// TwinCAT 3 PLC project PLC_1
// ProgramVersion: 3.1.4024.0
// libraries:
//   Tc2_MC2, * (Beckhoff Automation GmbH)
//   Tc2_Standard, * (Beckhoff Automation GmbH)
//   Tc2_System, * (Beckhoff Automation GmbH)
//   Tc3_IotBase, * (Beckhoff Automation GmbH)
//   Tc3_JsonXml, * (Beckhoff Automation GmbH)
//   Tc3_Module, * (Beckhoff Automation GmbH)
// project tree:
//   DUTs/ E_MC.TcDUT
//   GVLs/ GVL_PLC.TcGVL
//   / PlcTask.TcTTO
//   POUs/ FB_Sequence.TcPOU, FB_MQTT.TcPOU, MAIN.TcPOU
// real-time tasks:
//   TASK PlcTask: cycle T#10ms, priority 20, ADS port 350
// motion (NC):
//   TASK NC-Task 1 SAF: cycle T#2ms, priority 4, ADS port 501
//   TASK NC-Task 1 SVB: cycle T#10ms, priority 8, ADS port 511
//   AXIS StepAxis (id 1)
//     General: UnitName=Degree
//     Dynamic: Acceleration=727.2, Deceleration=727.2, Jerk=14689.4
//     Velo: Maximum=3600
//     PositionAreaControl: Enable=false
//     TargetPosControl: Enable=false
//     OtherSettings: AllowMotionCmdToSlave=true
//     encoder EncType=4
//       EncPara: ScaleFactorNumerator=0.028125, MaxCount=#x0000ffff
//         Inc: RefMode=2, RefSoftSyncMask=#x0000ffff
//     drive DrvType=24
//       Analog: VeloReferenz=3600, VeloScale=32, TorqueSetpointScale=10, ScaleFactorActTorque=0.1
//       TimeComp: TaskDelayCycles=1
//     controller CtrType=1
//       CtrPara: PriorControlFactor=1
//         PosDiffControl: Enable=false
//         PID: PosKp=3.5
//         Observer: BandWidth=20
//   AXIS Axis 2 (id 2)
//     OtherSettings: AllowMotionCmdToSlave=true
//     encoder EncType=4
//       EncPara: MaxCount=#x0000ffff
//         Inc: RefSoftSyncMask=#x0000ffff
//     drive DrvType=24
//       Analog: TorqueSetpointScale=10, ScaleFactorActTorque=0.1
//       TimeComp: TaskDelayCycles=1
//     controller CtrType=1
//       CtrPara: PriorControlFactor=1
//         Observer: BandWidth=20
//   AXIS ServoAxis (id 3)
//     General: UnitName=Degree
//     Dynamic: Acceleration=200, Deceleration=200, Jerk=100
//     Velo: Maximum=12000
//     PositionAreaControl: Enable=false
//     TargetPosControl: Enable=false
//     OtherSettings: AllowMotionCmdToSlave=true
//     encoder EncType=19
//       EncPara: ScaleFactorNumerator=0.000343322753906, MaxCount=#xffffffff
//     drive DrvType=16
//       DrvPara: MaxCount=#xffffffff, DriveControlDWord=#x00020000
//         Analog: VeloReferenz=12000, VeloScale=32, TorqueSetpointScale=10, ScaleFactorActTorque=0.1
//         TimeComp: TaskDelayCycles=1
//     controller CtrType=1
//       CtrPara: PriorControlFactor=1
//         PosDiffControl: Enable=false
//         Observer: BandWidth=20
// I/O:
//   DEVICE Device 3 (EtherCAT), AmsNetId 192.168.99.3.4.1
//     Term 1 (EK1100) [EK1100 EtherCAT Coupler (2A E-Bus)]
//       Term 2 (EL1008) [EL1008 8Ch. Dig. Input 24V, 3ms]
//       Term 3 (EL1008) [EL1008 8Ch. Dig. Input 24V, 3ms]
//       Term 4 (EL2008) [EL2008 8Ch. Dig. Output 24V, 0.5A]
//       Term 5 (EL2624) [EL2624 4Ch. Relay Output, NO (125V AC / 30V DC)]
//       Term 6 (EL6001) [EL6001 Interface (RS232)]
//       Term 15 (EL9011) [EL9011 End Terminal]
//     Term 7 (EK1100) [EK1100 EtherCAT Coupler (2A E-Bus)]
//       Term 8 (EL7031-0030) [EL7031-0030 1Ch. Stepper motor output stage (24V, 2.8A)]
//       Term 9 (EL6070-0033) [EL6070-0033 1Ch. Licence key terminal, individual licences]
//       Term 10 (EL7031-0030) [EL7031-0030 1Ch. Stepper motor output stage (24V, 2.8A)]
//       Term 16 (EL9011) [EL9011 End Terminal]
//     Term 11 (EK1818) [EK1818 EtherCAT IO-Coupler  (1A E-Bus, 8 Ch. Dig. In, 3ms, 4 Ch. Dig. Out 24V, 0,5A)]
//       Term 12 (EL7211-9014) [EL7211-9014 1Ch. MDP742 Servo motor output stage with OCT (50V, 4.5A RMS) and STO input]
//       Term 13 (EL1918) [EL1918, 8Ch. Safety Input 24V, TwinSAFE]
//         modules: Module 1 (FSOE), Module 2 (FSLOGIC)
//       Term 14 (EL3208) [EL3208 8Ch. Ana. Input PT100 (RTD)]
//       Term 17 (EL9011) [EL9011 End Terminal]
//   DEVICE Device 2 (RT-Ethernet Protocol), AmsNetId 192.168.99.3.3.1
// variable links:
//   NC-Task 1 SAF/Axes/Axis 2 <-> Device 3 (EtherCAT)/Term 7 (EK1100)/Term 10 (EL7031-0030)
//     Drive/Inputs/In/nState1 @bit 3 <-> STM Status/Status/Error
//     Drive/Inputs/In/nState1 @bit 5 <-> STM Status/Status/Moving negative
//     Drive/Inputs/In/nState1 @bit 4 <-> STM Status/Status/Moving positive
//     Drive/Inputs/In/nState1 @bit 1 <-> STM Status/Status/Ready
//     Drive/Inputs/In/nState1 <-> STM Status/Status/Ready to enable
//     Drive/Inputs/In/nState1 @bit 6 <-> STM Status/Status/Torque reduced
//     Drive/Inputs/In/nState1 @bit 2 <-> STM Status/Status/Warning
//     Drive/Inputs/In/nState2 @bit 3 <-> STM Status/Status/Digital input 1
//     Drive/Inputs/In/nState2 @bit 4 <-> STM Status/Status/Digital input 2
//     Drive/Inputs/In/nState2 @bit 5 <-> STM Status/Status/Sync error
//     Drive/Inputs/In/nState2 @bit 7 <-> STM Status/Status/TxPDO Toggle
//     Drive/Inputs/In/nState4 @bit 1 <-> WcState/InputToggle
//     Drive/Inputs/In/nState4 <-> WcState/WcState
//     Drive/Outputs/Out/nCtrl1 <-> STM Control/Control/Enable
//     Drive/Outputs/Out/nCtrl1 @bit 2 <-> STM Control/Control/Reduce torque
//     Drive/Outputs/Out/nCtrl1 @bit 1 <-> STM Control/Control/Reset
//     Drive/Outputs/Out/nDataOut2[0] <-> STM Velocity/Velocity
//     Enc/Inputs/In/nDataIn1[0] <-> ENC Status compact/Counter value
//     Enc/Inputs/In/nDataIn2[0] <-> ENC Status compact/Latch value
//     Enc/Inputs/In/nState1 @bit 4 <-> ENC Status compact/Status/Counter overflow
//     Enc/Inputs/In/nState1 @bit 3 <-> ENC Status compact/Status/Counter underflow
//     Enc/Inputs/In/nState1 @bit 1 <-> ENC Status compact/Status/Latch extern valid
//     Enc/Inputs/In/nState1 @bit 2 <-> ENC Status compact/Status/Set counter done
//     Enc/Inputs/In/nState2 @bit 4 <-> ENC Status compact/Status/Status of extern latch
//     Enc/Inputs/In/nState2 @bit 5 <-> ENC Status compact/Status/Sync error
//     Enc/Inputs/In/nState2 @bit 7 <-> ENC Status compact/Status/TxPDO Toggle
//     Enc/Inputs/In/nState4 @bit 1 <-> WcState/InputToggle
//     Enc/Inputs/In/nState4 <-> WcState/WcState
//     Enc/Outputs/Out/nCtrl1 @bit 3 <-> ENC Control compact/Control/Enable latch extern on negative edge
//     Enc/Outputs/Out/nCtrl1 @bit 1 <-> ENC Control compact/Control/Enable latch extern on positive edge
//     Enc/Outputs/Out/nCtrl1 @bit 2 <-> ENC Control compact/Control/Set counter
//     Enc/Outputs/Out/nDataOut1[0] <-> ENC Control compact/Set counter value
//   NC-Task 1 SAF/Axes/ServoAxis <-> Device 3 (EtherCAT)/Term 11 (EK1818)/Term 12 (EL7211-9014)
//     Drive/Inputs/In/nDcOutputTime <-> InfoData/DcOutputShift
//     Drive/Inputs/In/nState1 <-> DRV Statusword/Statusword
//     Drive/Inputs/In/nState2 <-> DRV Statusword/Statusword @bit 8
//     Drive/Inputs/In/nState4 @bit 1 <-> WcState/InputToggle
//     Drive/Inputs/In/nState4 <-> WcState/WcState
//     Drive/Outputs/Out/nCtrl1 <-> DRV Controlword/Controlword
//     Drive/Outputs/Out/nCtrl2 <-> DRV Controlword/Controlword @bit 8
//     Drive/Outputs/Out/nDataOut2 <-> DRV Target velocity/Target velocity
//     Enc/Inputs/In/nDataIn1 <-> FB Position/Position
//     Enc/Inputs/In/nDcInputTime <-> InfoData/DcInputShift
//     Enc/Inputs/In/nState4 @bit 1 <-> WcState/InputToggle
//     Enc/Inputs/In/nState4 <-> WcState/WcState
//   NC-Task 1 SAF/Axes/StepAxis <-> Device 3 (EtherCAT)/Term 7 (EK1100)/Term 8 (EL7031-0030)
//     Drive/Inputs/In/nState1 @bit 3 <-> STM Status/Status/Error
//     Drive/Inputs/In/nState1 @bit 5 <-> STM Status/Status/Moving negative
//     Drive/Inputs/In/nState1 @bit 4 <-> STM Status/Status/Moving positive
//     Drive/Inputs/In/nState1 @bit 1 <-> STM Status/Status/Ready
//     Drive/Inputs/In/nState1 <-> STM Status/Status/Ready to enable
//     Drive/Inputs/In/nState1 @bit 6 <-> STM Status/Status/Torque reduced
//     Drive/Inputs/In/nState1 @bit 2 <-> STM Status/Status/Warning
//     Drive/Inputs/In/nState2 @bit 3 <-> STM Status/Status/Digital input 1
//     Drive/Inputs/In/nState2 @bit 4 <-> STM Status/Status/Digital input 2
//     Drive/Inputs/In/nState2 @bit 5 <-> STM Status/Status/Sync error
//     Drive/Inputs/In/nState2 @bit 7 <-> STM Status/Status/TxPDO Toggle
//     Drive/Inputs/In/nState4 @bit 1 <-> WcState/InputToggle
//     Drive/Inputs/In/nState4 <-> WcState/WcState
//     Drive/Outputs/Out/nCtrl1 <-> STM Control/Control/Enable
//     Drive/Outputs/Out/nCtrl1 @bit 2 <-> STM Control/Control/Reduce torque
//     Drive/Outputs/Out/nCtrl1 @bit 1 <-> STM Control/Control/Reset
//     Drive/Outputs/Out/nDataOut2[0] <-> STM Velocity/Velocity
//     Enc/Inputs/In/nDataIn1[0] <-> ENC Status compact/Counter value
//     Enc/Inputs/In/nDataIn2[0] <-> ENC Status compact/Latch value
//     Enc/Inputs/In/nState1 @bit 4 <-> ENC Status compact/Status/Counter overflow
//     Enc/Inputs/In/nState1 @bit 3 <-> ENC Status compact/Status/Counter underflow
//     Enc/Inputs/In/nState1 @bit 1 <-> ENC Status compact/Status/Latch extern valid
//     Enc/Inputs/In/nState1 @bit 2 <-> ENC Status compact/Status/Set counter done
//     Enc/Inputs/In/nState2 @bit 4 <-> ENC Status compact/Status/Status of extern latch
//     Enc/Inputs/In/nState2 @bit 5 <-> ENC Status compact/Status/Sync error
//     Enc/Inputs/In/nState2 @bit 7 <-> ENC Status compact/Status/TxPDO Toggle
//     Enc/Inputs/In/nState4 @bit 1 <-> WcState/InputToggle
//     Enc/Inputs/In/nState4 <-> WcState/WcState
//     Enc/Outputs/Out/nCtrl1 @bit 3 <-> ENC Control compact/Control/Enable latch extern on negative edge
//     Enc/Outputs/Out/nCtrl1 @bit 1 <-> ENC Control compact/Control/Enable latch extern on positive edge
//     Enc/Outputs/Out/nCtrl1 @bit 2 <-> ENC Control compact/Control/Set counter
//     Enc/Outputs/Out/nDataOut1[0] <-> ENC Control compact/Set counter value
//   PLC_1/PLC_1 Instance <-> Device 2 (RT-Ethernet Protocol)
//     PlcTask Inputs/GVL_PLC.uiDevState <-> Inputs/DevState
//   PLC_1/PLC_1 Instance <-> Device 3 (EtherCAT)/Term 1 (EK1100)/Term 2 (EL1008)
//     PlcTask Inputs/MAIN.fbSequence.xButton_NO3 <-> Channel 1/Input
//   PLC_1/PLC_1 Instance <-> Device 3 (EtherCAT)/Term 1 (EK1100)/Term 3 (EL1008)
//     PlcTask Inputs/MAIN.fbSequence.xButton_NO1 <-> Channel 2/Input
//     PlcTask Inputs/MAIN.fbSequence.xButton_NO2 <-> Channel 7/Input
//   PLC_1/PLC_1 Instance <-> NC-Task 1 SAF/Axes/ServoAxis
//     PlcTask Inputs/MAIN.ServoAxis.NcToPlc <-> Outputs/ToPlc
//     PlcTask Outputs/MAIN.ServoAxis.PlcToNc <-> Inputs/FromPlc
//   PLC_1/PLC_1 Instance <-> NC-Task 1 SAF/Axes/StepAxis
//     PlcTask Inputs/MAIN.StepAxis.NcToPlc <-> Outputs/ToPlc
//     PlcTask Outputs/MAIN.StepAxis.PlcToNc <-> Inputs/FromPlc

CONFIGURATION PLC_1
    RESOURCE PLC ON TwinCAT3
        TASK PlcTask(INTERVAL := T#10ms, PRIORITY := 20);
        PROGRAM MAIN WITH PlcTask : MAIN;
    END_RESOURCE
END_CONFIGURATION

// ---- DUTs/E_MC.TcDUT
{attribute 'qualified_only'}
{attribute 'strict'}
TYPE E_MC :
(
	Idle,
	
	RestartCall,
	RestartEffect,
	PowerCall,
	PowerEffect,
	
	HomingCallStep,   
	HomingEffectStep,
	HomingCallServo,   
	HomingEffectServo,
	Execute,
	
	CoupleCallStepMaster,
	CoupleEffectStepMaster,
	MoveAbsCallStepMaster,
	MoveAbsEffectStepMaster,
	DecoupleCallStepMaster,
	DecoupleEffectStepMaster,
	
	
	CoupleCallServoMaster,
	CoupleEffectServoMaster,
	MoveAbsCallServoMaster,
	MoveAbsEffectServoMaster,
	DecoupleCallServoMaster,
	DecoupleEffectServoMaster,
	
	DecoupleCallOnReset,
	DecoupleEffectOnReset,	
	RestartCallOnReset,
	RestartEffectOnReset,	
	
	Error
);
END_TYPE

// ---- GVLs/GVL_PLC.TcGVL
{attribute 'qualified_only'}
VAR_GLOBAL
	lrActPosition	:	LREAL;
	uiDevState	AT%I*	:	UINT;
END_VAR

// ---- POUs/MAIN.TcPOU
PROGRAM MAIN
VAR
	StepAxis	:	AXIS_REF;
	ServoAxis	:	AXIS_REF;
	fbMqtt		:	FB_MQTT;
	fbSequence	:	FB_Sequence;
END_VAR


fbMqtt();
GVL_PLC.lrActPosition := ServoAxis.NcToPlc.ActPos;

fbSequence(ServoAxis:=ServoAxis,StepAxis:=StepAxis);

ServoAxis();
StepAxis();

END_PROGRAM

// ---- POUs/FB_MQTT.TcPOU
FUNCTION_BLOCK FB_MQTT
VAR
		//MQTT
	sBrokerIP	: 			STRING:='192.168.8.101';	// Beckhoff IP
	uiPortNumber:			UINT:=1883;				// Port using for mqtt exchange 
	sPrefix		:			STRING:='MQTT/cseg';	// Prefix of mqtt server
	sTopic		:			STRING:='/PositionOfMotor';	// Topic in which our variable is being saved 
	bInitialize :			BOOL;
	bConnect	:			BOOL;
	
	// MQTT Function Blocks 
	fbMQTTClient	:		FB_IotMqttClient;
	fbMQTTMessage	:		FB_IotMqttMessage;
	fbMQTTMessageQueue:		FB_IotMqttMessageQueue;
	
	tonPublishingData	:	TON;
	sMessage		:		STRING;
	
	bRetain:BOOL;
	bQueue:BOOL;
END_VAR

// Setting variables for connection
IF bInitialize THEN
	bInitialize:=FALSE;
	fbMQTTClient.sHostName := sBrokerIP;
	fbMQTTClient.nHostPort := uiPortNumber;
	fbMQTTClient.sTopicPrefix := sPrefix;
	fbMQTTClient.ipMessageQueue := fbMQTTMessageQueue;
	
 	bConnect := TRUE;
END_IF

fbMQTTClient.Execute(bConnect);

IF fbMQTTClient.bConnected THEN
	tonPublishingData(IN:= NOT tonPublishingData.Q , PT:=T#3S); // Publishing every 1s
	IF tonPublishingData.Q THEN
		sMessage := CONCAT('Motor Position: ',LREAL_TO_STRING(GVL_PLC.lrActPosition)); 	// Writing motor Position into broker
		fbMQTTClient.Publish(
					sTopic:=sTopic , 
					nPayloadSize:=INT_TO_UDINT(LEN(sMessage)) , 
					pPayload:=ADR(sMessage) , 
					eQoS:= TcIotMqttQos.AtLeastOnceDelivery , 
					bRetain:=FALSE , 
					bQueue:=FALSE );
	END_IF
END_IF

END_FUNCTION_BLOCK

// ---- POUs/FB_Sequence.TcPOU
FUNCTION_BLOCK FB_Sequence
VAR_IN_OUT
	ServoAxis	:	AXIS_REF;			// Axises of two motors
	StepAxis	:	AXIS_REF;
END_VAR
VAR
	Slave		:	AXIS_REF;			// Slave and master axises
	Master		:	AXIS_REF;
	fbGearIn	:	MC_GearIn;			// Motion control function blocks
	fbMoveAbsolute	:	MC_MoveAbsolute;
	fbGearOut	:	MC_GearOut;
	fbResetServo 	: 			MC_Reset;
	fbResetStep 	: 			MC_Reset;
	fbPowerServo 	: 			MC_Power;
	xGearIn		:	BOOL;				// Coupling motors
	xGearOut	:	BOOL;				// Decoupling motors
    lrRatioNumerator   : LREAL:=1;
    uiRatioDenominator : UINT:=1;
	fbPowerStep	: 			MC_Power;
	xManualReset	 : 		BOOL; // Resetting program
	xPowerOn	:			BOOL; //Enabling power sources
	xExecute	:			BOOL; // Executing program
	eStateMc 	: 			E_MC ;//instance of enum
	eStatePrevious	:		E_MC;
	xStepIsMaster		:		BOOL;
	xStepIsSlave	:		BOOL;
	lrPosition	: 			LREAL; 	//Target Position
	lrVelocity 	:			LREAL; 	// Setting Velocity
	lrRealPosition:			LREAL;	// real position
	xButton_NO1 	AT%I* : BOOL;
	xButton_NO2 	AT%I* : BOOL;
	xButton_NO3		AT%I* : BOOL;
	fTriggerStart			:	F_TRIG;
	fTriggerReset			:	F_TRIG;		// Falling triggers on 3 buttons
	fTriggerHome			:	F_TRIG;
	xStartSequence		:	BOOL;			// starting sequence
	xResetErrors		:	BOOL;			// Reseting errors
	xHomeMotors				:	BOOL;		// Homing motors
	tonTooLongInCase	:	TON;			// Ton timer counting time in each case
	xTooLongInCase		:	BOOL;		   // Too long in case
	sErrorLocalization	:	STRING(255);  // Moment when error occured
END_VAR

fTriggerStart(CLK:=xButton_NO2 , Q=>xStartSequence );		// Triggers on buttons
fTriggerReset(CLK:=xButton_NO1 , Q=>xResetErrors );
fTriggerHome(CLK:=xButton_NO3 , Q=>xHomeMotors );
lrRealPosition:=ServoAxis.NcToPlc.ActPos;
// Timer in each case
IF (eStateMc <> E_MC.Idle) AND (eStateMc <> E_MC.Error)  THEN
	IF eStateMc <> eStatePrevious THEN			// Comparing  current and previous values of enum
		tonTooLongInCase(IN := FALSE); 			// Reseting clock
		eStatePrevious := eStateMc; 			// timeout string
	END_IF

	tonTooLongInCase(IN := TRUE, PT :=T#20S);
	
	IF tonTooLongInCase.Q THEN
		eStateMc := E_MC.Error; 
		sErrorLocalization:='Timeout';
	END_IF
END_IF
// Case of program states
CASE eStateMc OF
	
	E_MC.Idle:									// Start of the program, homing
		IF xHomeMotors THEN
			xHomeMotors:=FALSE;
			eStateMc:=E_MC.RestartCall;
		END_IF
		
	E_MC.RestartCall:							// Calling reset of the errors
		xManualReset:=TRUE;							
		IF fbResetServo.Busy AND fbResetStep.Busy THEN
				eStateMc:=E_MC.RestartEffect;					
		ELSIF	fbResetServo.Error OR fbResetStep.Error THEN
			eStateMc:=E_MC.Error;
			sErrorLocalization:='Error when reseting motor errors(RestartCall)';
		END_IF
		
	E_MC.RestartEffect:						// Executing reset 
		xManualReset:=FALSE;
		IF fbResetServo.Done AND fbResetStep.Done THEN
			eStateMc:=E_MC.PowerCall;
		ELSIF	fbResetServo.Error OR fbResetStep.Error THEN
			eStateMc:=E_MC.Error;
			sErrorLocalization:='Error when reseting motor errors(RestartEffect)';
		END_IF
		
	E_MC.PowerCall:								// Calling power enable
		xPowerOn:=TRUE;
		IF fbPowerServo.Busy AND fbPowerStep.Busy THEN
				eStateMc:=E_MC.PowerEffect;
		ELSIF	fbPowerServo.Error OR fbPowerStep.Error THEN
			eStateMc:=E_MC.Error;
			sErrorLocalization:='Error when enabling motors power(PowerCall)';
		END_IF
		
	E_MC.PowerEffect:
		IF fbPowerServo.Status AND fbPowerStep.Status THEN
			eStateMc:=E_MC.HomingCallServo;
		ELSIF	fbPowerServo.Error OR fbPowerStep.Error THEN
			eStateMc:=E_MC.Error;
			sErrorLocalization:='Error when enabling motors power(PowerEffect)';
		END_IF
	
	E_MC.HomingCallServo:			// Homing servo motor
		Master:=ServoAxis;
		lrPosition:=0;
		lrVelocity:=100;
		xExecute:=TRUE;
		IF fbMoveAbsolute.Busy THEN
			eStateMc := E_MC.HomingEffectServo;
		END_IF
		IF fbMoveAbsolute.Error THEN
			// Going into error step, when error id is 1800 write information about it
			eStateMc:=E_MC.Error;
			IF ServoAxis.Status.ErrorID=16#00004650 THEN
				sErrorLocalization:=CONCAT(CONCAT('Error homing servo motor(HomingCallStep) ErrorID: ',UDINT_TO_STRING(ServoAxis.Status.ErrorID)),' Drive hardware not ready to operate');
			ELSE
				sErrorLocalization:='Error homing servo motor(HomingCallStep)';
			END_IF
		END_IF
		
	E_MC.HomingEffectServo:
		Master:=ServoAxis;
		xExecute:=FALSE;
		IF fbMoveAbsolute.Done THEN
			eStateMc:=E_MC.HomingCallStep;
		END_IF

		IF fbMoveAbsolute.Error THEN
			eStateMc:=E_MC.Error;
			IF ServoAxis.Status.ErrorID=16#00004650 THEN
				sErrorLocalization:=CONCAT(CONCAT('Error homing servo motor(HomingEffectServo) ErrorID: ',UDINT_TO_STRING(ServoAxis.Status.ErrorID)),' Drive hardware not ready to operate');
			ELSE
				sErrorLocalization:='Error homing servo motor(HomingEffectServo)';
			END_IF
		END_IF	

	E_MC.HomingCallStep:			// Homing Step motor
		Master:=StepAxis;
		lrPosition:=0;
		lrVelocity:=100;
		xExecute:=TRUE;
		IF fbMoveAbsolute.Busy THEN
			eStateMc := E_MC.HomingEffectStep;
		END_IF
		IF fbMoveAbsolute.Error THEN
			eStateMc:=E_MC.Error;
			IF StepAxis.Status.ErrorID=16#00004650 THEN
				sErrorLocalization:=CONCAT(CONCAT('Error homing servo motor(HomingCallStep) ErrorID: ',UDINT_TO_STRING(StepAxis.Status.ErrorID)),' Drive hardware not ready to operate');
			ELSE
				sErrorLocalization:='Error homing step motor(HomingCallStep)';
			END_IF			
		END_IF
		
	E_MC.HomingEffectStep:
		Master:=StepAxis;
		xExecute:=FALSE;
		IF fbMoveAbsolute.Done THEN
			eStateMc:=E_MC.Execute;
		END_IF

		IF fbMoveAbsolute.Error THEN
			eStateMc:=E_MC.Error;
			IF StepAxis.Status.ErrorID=16#00004650 THEN
				sErrorLocalization:=CONCAT(CONCAT('Error homing servo motor(HomingEffectStep) ErrorID: ',UDINT_TO_STRING(StepAxis.Status.ErrorID)),' Drive hardware not ready to operate');
			ELSE
				sErrorLocalization:='Error homing step motor(HomingEffectStep)';
			END_IF	
		END_IF		
	// Waiting for start button 
	E_MC.Execute:
		IF 	xStartSequence THEN
			xStartSequence:=FALSE;
			eStateMc:=E_MC.CoupleCallStepMaster;
		END_IF
		
	E_MC.CoupleCallStepMaster:					// Coupling Motors
		IF ServoAxis.Status.Coupled THEN
		eStateMc:=E_MC.MoveAbsCallStepMaster;
		END_IF
		Master := StepAxis;
		Slave  := ServoAxis;
		xGearIn:=TRUE;
		IF fbGearIn.Busy THEN
			eStateMc:=E_MC.CoupleEffectStepMaster;
		END_IF								
		IF fbGearIn.Error THEN
			eStateMc:=E_MC.Error;
			sErrorLocalization:='Error coupling motors(CoupleCallStepMaster)';
		END_IF
		
	E_MC.CoupleEffectStepMaster:
		IF fbGearIn.InGear  THEN
			eStateMc:=E_MC.MoveAbsCallStepMaster;
		ELSIF fbGearIn.Error THEN
			eStateMc:=E_MC.Error;
			sErrorLocalization:='Error coupling motors(CoupleEffectStepMaster)';
		END_IF	
	
	E_MC.MoveAbsCallStepMaster:				// move absolute for first coupling
		Master:=StepAxis;
		lrPosition:=720;
		lrVelocity:=100;
		xExecute:=TRUE;
		IF fbMoveAbsolute.Busy THEN
			eStateMc := E_MC.MoveAbsEffectStepMaster;
		END_IF
		IF fbMoveAbsolute.Error THEN
			eStateMc:=E_MC.Error;
			IF StepAxis.Status.ErrorID=16#00004650 THEN
				sErrorLocalization:=CONCAT(CONCAT('Error in step motor movement(MoveAbsCallStepMaster) ErrorID: ',UDINT_TO_STRING(StepAxis.Status.ErrorID)),' Drive hardware not ready to operate');
			ELSIF ServoAxis.Status.ErrorID=16#00004650 THEN
				sErrorLocalization:=CONCAT(CONCAT('Error in servo motor movement(MoveAbsCallStepMaster) ErrorID: ',UDINT_TO_STRING(ServoAxis.Status.ErrorID)),' Drive hardware not ready to operate');
			ELSE
				sErrorLocalization:='Error in motors movement(MoveAbsCallStepMaster)';
			END_IF	
		END_IF
		
	E_MC.MoveAbsEffectStepMaster:
		Master:=StepAxis;
		xExecute:=FALSE;
		IF fbMoveAbsolute.Done THEN
			eStateMc:=E_MC.DecoupleCallStepMaster;
		END_IF

		IF fbMoveAbsolute.Error THEN
			eStateMc:=E_MC.Error;
			IF StepAxis.Status.ErrorID=16#00004650 THEN
				sErrorLocalization:=CONCAT(CONCAT('Error in step motor movement(MoveAbsEffectStepMaster) ErrorID: ',UDINT_TO_STRING(StepAxis.Status.ErrorID)),' Drive hardware not ready to operate');
			ELSIF ServoAxis.Status.ErrorID=16#00004650 THEN
				sErrorLocalization:=CONCAT(CONCAT('Error in servo motor movement(MoveAbsEffectStepMaster) ErrorID: ',UDINT_TO_STRING(ServoAxis.Status.ErrorID)),' Drive hardware not ready to operate');
			ELSE
				sErrorLocalization:='Error in motors movement(MoveAbsEffectStepMaster)';
			END_IF	
		END_IF	
	
	E_MC.DecoupleCallStepMaster:				// Decoupling motors
		xGearIn:=FALSE;
		xGearOut:=TRUE;
		Slave:=ServoAxis;
		IF fbGearOut.Busy THEN
			eStateMc:=E_MC.DecoupleEffectStepMaster;		
		ELSIF fbGearOut.Error THEN
			eStateMc:=E_MC.Error;
			sErrorLocalization:='Error decoupling motors(DecoupleCallStepMaster)';
		END_IF	
		
	E_MC.DecoupleEffectStepMaster:
		xGearOut:=FALSE;
		Slave:=ServoAxis;
		IF fbGearOut.Done  THEN
			eStateMc:=E_MC.CoupleCallServoMaster;
		ELSIF fbGearOut.Error THEN
			eStateMc:=E_MC.Error;
			sErrorLocalization:='Error decoupling motors(DecoupleEffectStepMaster)';
		END_IF	
		
	E_MC.CoupleCallServoMaster:						// Second couple 
		IF StepAxis.Status.Coupled THEN
		eStateMc:=E_MC.MoveAbsCallServoMaster;
		END_IF
		
		Master := ServoAxis;
		Slave  := StepAxis;
		xGearIn:=TRUE;
		IF fbGearIn.Busy THEN
			eStateMc:=E_MC.CoupleEffectServoMaster;
		END_IF								
		IF fbGearIn.Error THEN
			eStateMc:=E_MC.Error;
			sErrorLocalization:='Error coupling motors(CoupleCallServoMaster)';
		END_IF	

	E_MC.CoupleEffectServoMaster:
		IF fbGearIn.InGear  THEN
			eStateMc:=E_MC.MoveAbsCallServoMaster;
		ELSIF fbGearIn.Error THEN
			eStateMc:=E_MC.Error;
			sErrorLocalization:='Error coupling motors(CoupleEffectServoMaster)';
		END_IF	

	E_MC.MoveAbsCallServoMaster:				// Move absolute for second couple
		Master := ServoAxis;
		lrPosition:=0;
		lrVelocity:=100;
		xExecute:=TRUE;
		IF fbMoveAbsolute.Busy THEN
			eStateMc := E_MC.MoveAbsEffectServoMaster;
		END_IF
		IF fbMoveAbsolute.Error THEN 
			eStateMc:=E_MC.Error;
			IF StepAxis.Status.ErrorID=16#00004650 THEN
				sErrorLocalization:=CONCAT(CONCAT('Error in step motor movement(MoveAbsCallServoMaster) ErrorID: ',UDINT_TO_STRING(StepAxis.Status.ErrorID)),' Drive hardware not ready to operate');
			ELSIF ServoAxis.Status.ErrorID=16#00004650 THEN
				sErrorLocalization:=CONCAT(CONCAT('Error in servo motor movement(MoveAbsCallServoMaster) ErrorID: ',UDINT_TO_STRING(ServoAxis.Status.ErrorID)),' Drive hardware not ready to operate');
			ELSE
				sErrorLocalization:='Error in motors movement(MoveAbsCallServoMaster)';
			END_IF	
		END_IF
	
	E_MC.MoveAbsEffectServoMaster:
		Master:=ServoAxis;
		xExecute:=FALSE;
		IF fbMoveAbsolute.Done THEN
			eStateMc:=E_MC.DecoupleCallServoMaster;
		END_IF
		
		IF fbMoveAbsolute.Error THEN
			eStateMc:=E_MC.Error;
			IF StepAxis.Status.ErrorID=16#00004650 THEN
				sErrorLocalization:=CONCAT(CONCAT('Error in step motor movement(MoveAbsEffectServoMaster) ErrorID: ',UDINT_TO_STRING(StepAxis.Status.ErrorID)),' Drive hardware not ready to operate');
			ELSIF ServoAxis.Status.ErrorID=16#00004650 THEN
				sErrorLocalization:=CONCAT(CONCAT('Error in servo motor movement(MoveAbsEffectServoMaster) ErrorID: ',UDINT_TO_STRING(ServoAxis.Status.ErrorID)),' Drive hardware not ready to operate');
			ELSE
				sErrorLocalization:='Error in motors movement(MoveAbsEffectServoMaster)';
			END_IF	
		END_IF					
	
	E_MC.DecoupleCallServoMaster:				// Decoupling
		xGearIn:=FALSE;
		xGearOut:=TRUE;
		Slave:=StepAxis;
		IF fbGearOut.Busy THEN
			eStateMc:=E_MC.DecoupleEffectServoMaster;		
		ELSIF fbGearOut.Error THEN
			eStateMc:=E_MC.Error;
			sErrorLocalization:='Error decoupling motors(DecoupleCallServoMaster)';
		END_IF	
		
		
	E_MC.DecoupleEffectServoMaster:
		xGearOut:=FALSE;
		Slave:=StepAxis;
		IF fbGearOut.Done  THEN
			eStateMc:=E_MC.Idle;
		ELSIF fbGearOut.Error THEN
			eStateMc:=E_MC.Error;
			sErrorLocalization:='Error decoupling motors(DecoupleEffectServoMaster)';
		END_IF		
	
		
	// Cases for when error occurs 	
		
	E_MC.DecoupleCallOnReset:							// Decoupling after reset
		IF StepAxis.Status.Coupled THEN
			Slave:=StepAxis;
		ELSIF ServoAxis.Status.Coupled THEN
			Slave:=ServoAxis;
		END_IF
		xGearIn:=FALSE;
		xGearOut:=TRUE;
		IF fbGearOut.Busy THEN
			eStateMc:=E_MC.DecoupleEffectOnReset;		
		ELSIF fbGearOut.Error THEN
			eStateMc:=E_MC.Error;
			sErrorLocalization:='Error decoupling motors(DecoupleCallOnReset)';
		END_IF	
	
	E_MC.DecoupleEffectOnReset:	
		IF StepAxis.Status.Coupled THEN
			Slave:=StepAxis;
		ELSIF ServoAxis.Status.Coupled THEN
			Slave:=ServoAxis;
		END_IF
		xGearOut:=FALSE;
		Slave:=StepAxis;
		IF fbGearOut.Done  THEN
			eStateMc:=E_MC.RestartCallOnReset;
		ELSIF fbGearOut.Error THEN
			eStateMc:=E_MC.Error;
			sErrorLocalization:='Error decoupling motors(DecoupleEffectOnReset)';
		END_IF		
		
	E_MC.RestartCallOnReset:									// Reseting errors after reset 
		xManualReset:=TRUE;							
		IF fbResetServo.Busy AND fbResetStep.Busy THEN
				eStateMc:=E_MC.RestartEffectOnReset;					
		ELSIF	fbResetServo.Error OR fbResetStep.Error THEN
			eStateMc:=E_MC.Error;
			sErrorLocalization:='Error when reseting motor errors(RestartCallOnReset)';
		END_IF
		
	E_MC.RestartEffectOnReset:	
		xManualReset:=FALSE;
		IF fbResetServo.Done AND fbResetStep.Done THEN
			eStateMc:=E_MC.Idle;
		ELSIF	fbResetServo.Error OR fbResetStep.Error THEN
			eStateMc:=E_MC.Error;
			sErrorLocalization:='Error when reseting motor errors(RestartEffectOnReset)';
		END_IF
		
	E_MC.Error:									// Error case, turning power off and going to next case
		xPowerOn:=FALSE;
		IF xResetErrors THEN
			xResetErrors:=FALSE;
			sErrorLocalization:='';
			IF StepAxis.Status.Coupled OR ServoAxis.Status.Coupled THEN
				eStateMc := E_MC.DecoupleCallOnReset;
			ELSE
				eStateMc := E_MC.RestartCallOnReset;
			END_IF	
		END_IF
END_CASE


//SERVO MOTOR
fbResetServo(				//Reseting motor // Reset1 -> ResetServoMotor
	Axis:= ServoAxis, 
	Execute:= xManualReset, 
	Done=> , 
	Busy=> , 
	Error=> , 
	ErrorID=> );
	
fbPowerServo(				// Turning power on
	Axis:= ServoAxis, 
	Enable:= xPowerOn, 
	Enable_Positive:= xPowerOn, 
	Enable_Negative:= xPowerOn, 
	Override:= 100, 
	BufferMode:= , 
	Options:= , 
	Status=> , 
	Busy=> , 
	Error=> , 
	ErrorID=> );
	
	
//STEP MOTOR
fbResetStep(				//Reseting motor
	Axis:= StepAxis, 
	Execute:= xManualReset, 
	Done=> , 
	Busy=> , 
	Error=> , 
	ErrorID=> );
	
fbPowerStep(				// Turning power on
	Axis:= StepAxis, 
	Enable:= xPowerOn, 
	Enable_Positive:= xPowerOn, 
	Enable_Negative:= xPowerOn, 
	Override:= 100, 
	BufferMode:= , 
	Options:= , 
	Status=> , 
	Busy=> , 
	Error=> , 
	ErrorID=> );
	
	
fbMoveAbsolute(			// Executing program
	Axis:= Master, 
	Execute:= xExecute, 
	Position:=lrPosition, 
	Velocity:= lrVelocity, 
	Acceleration:= , 
	Deceleration:= , 
	Jerk:= , 
	BufferMode:= , 
	Options:= , 
	Done=> , 
	Busy=> , 
	Active=> , 
	CommandAborted=> , 
	Error=> , 
	ErrorID=> );
fbGearIn(
		Master:=Master , 
		Slave:=Slave , 
		Execute:=xGearIn , 
		RatioNumerator:=lrRatioNumerator , 
		RatioDenominator:= uiRatioDenominator, 
		Acceleration:= , 
		Deceleration:= , 
		Jerk:= , 
		BufferMode:= , 
		Options:= , 
		InGear=> , 
		Busy=> , 
		Active=> , 
		CommandAborted=> , 
		Error=> , 
		ErrorID=> );
	
fbGearOut(
		Slave:= Slave, 
		Execute:=xGearOut , 
		Options:= , 
		Done=> , 
		Busy=> , 
		Error=> , 
		ErrorID=> );

END_FUNCTION_BLOCK
